{attribute 'qualified_only'}
{attribute 'strict'}
TYPE RESPONSE_STATE :
(
	UNDEFINED,
	BUSY,
	DONE,
	DONE_PENDING,
	SUBSTATE,
	ERROR,
	NO_IMPL
);
END_TYPE

(* stored: Version 1.1.0.1
   EnumerationTextList RESPONSE_STATE: Id {004c55da-6eec-4679-a40a-9d699817a4f2} *)
